// TIA Portal project "PLC_stage_DIPLOMA" (V19)

(* hardware
DEVICE "S7-1500/ET200MP station_1"  S7-1500 station
   slot 0: "Rail_0"  Rack  6ES7 590-1***0-0AA0
   slot 1: "PLC_1"  CPU 1513F-1 PN  6ES7 513-1FL02-0AB0  V2.9
      slot 3: "CPU display_1"  6ES7591-1AA00-0AA0
      slot 32768: "PROFINET interface_1"  X1
      slot 34817: "Virtual CP interface port_1"  Virtual CP interface port  Virtual CP interface port
   slot 2: "DI 32x24VDC HF_1"  DI 32x24VDC HF  6ES7 521-1BL00-0AB0  V2.2
   slot 3: "DQ 32x24VDC/0.5A HF_1"  DQ 32x24VDC/0.5A HF  6ES7 522-1BL01-0AB0  V1.1
   slot 4: "AI 8xU/I/RTD/TC ST_1"  AI 8xU/I/RTD/TC ST  6ES7 531-7KF00-0AB0  V2.2
DEVICE "ET 200SP station_1"  ET 200SP-Station
   slot 0: "Rack_0"  Rack  6ES5 710-8MAx1
   slot 0: "IO device_1"  IM 155-6 PN ST  6ES7 155-6AU01-0BN0  V4.2
   slot 1: "DI 8x24VDC ST_1"  DI 8x24VDC ST  6ES7 131-6BF01-0BA0  V0.0
      slot 1: "DI 8x24VDC ST_1"  DI 8x24VDC ST
   slot 2: "DI 8x24VDC ST_2"  DI 8x24VDC ST  6ES7 131-6BF01-0BA0  V0.0
      slot 1: "DI 8x24VDC ST_2"  DI 8x24VDC ST
   slot 3: "DQ 16x24VDC/0.5A ST_1"  DQ 16x24VDC/0.5A ST  6ES7 132-6BH01-0BA0  V0.0
      slot 1: "DQ 16x24VDC/0.5A ST_1"  DQ 16x24VDC/0.5A ST
   slot 4: "AI 4xU/I 2-wire ST_2"  AI 4xU/I 2-wire ST  6ES7 134-6HD01-0BA1  V2.0
      slot 1: "AI 4xU/I 2-wire ST_2"  AI 4xU/I 2-wire ST
   slot 5: "AQ 4xU/I ST_1"  AQ 4xU/I ST  6ES7 135-6HD00-0BA1  V1.1
      slot 1: "AQ 4xU/I ST_1"  AQ 4xU/I ST
   slot 6: "Server module_1"  Server module  6ES7 193-6PA00-0AA0  V1.1
      slot 1: "Server module_1"  Server module
   slot 127: "BA 2xRJ45"  BA 2xRJ45  6ES7 193-6AR00-0AA0  V0.0
      slot 1: "Port_1"  X1 P1 R  6ES7 193-6AR00-0AA0  V0.0
      slot 2: "Port_2"  X1 P2 R  6ES7 193-6AR00-0AA0  V0.0
DEVICE "PC-System_1"  SIMATIC PC station
   slot 0: "SIMATIC PC station"  Rail  SIMATIC PC-Station  V1.0
      slot 125: "Stationmanager"  Station_Manager  V6.0.4
   slot 1: "HMI_RT_2"  WinCC RT Advanced  6AV2 104-0xxxx-xxxx  17.0.0.0
      slot 33792: "Computer interface"  Host interface
   slot 2: "IE general_1"  IE General  IE_CP  V8.2.0
      slot 1: "PROFINET interface"  IEGeneral.Interface.8.2.0
DEVICE "HMI_1"  TP700 Comfort
   slot 0: "HMI_1"  TP700 Comfort  6AV2 124-0GC01-0AX0  17.0.0.0
   slot 1: "HMI_RT_1"  TP700 Comfort  6AV2 124-0GC01-0AX0  17.0.0.0
   slot 5: "HMI_1.IE_CP_1"  PROFINET Interface  17.0.0.0
      slot 1: "PROFINET Interface_1"  PROFINET Interface
         slot 1: "Port_1"  Port
         slot 2: "Port_2"  Port
   slot 7: "HMI_1.MPI/DP_CP_1"  MPI/DP Interface  17.0.0.0
*)

// ===== PLC "PLC_1"  CPU 1513F-1 PN =====

VAR_GLOBAL   // PLC tag table "additional_variables"
   "Get_value1_from_Matlab" AT %M11.0 : Bool;
   "AlwaysFALSE" AT %M0.3 : Bool;
   "Get_value2_from_Matlab" AT %M11.1 : Bool;
   "Send_value1_to_Matlab" AT %M11.2 : Bool;
   "Send_value2_to_Matlab" AT %M11.4 : Bool;
   "HMI_FN101_Visible1" AT %Q1.1 : Bool;
   "HMI_FN101_Visible2" AT %Q1.2 : Bool;
   "HMI_RB102_Visible" AT %Q1.4 : Bool;
   "HMI_WP101_Painted" AT %Q1.6 : Bool;
   "HMI_WP101_Visible" AT %M7.0 : Bool;
   "HMI_WP102_Visible" AT %M7.1 : Bool;
   "HMI_WP103_Visible" AT %M7.2 : Bool;
   "HMI_WP104_Visible" AT %M7.3 : Bool;
   "HMI_Main" AT %M7.4 : Bool;
   "HMI_PID" AT %M7.5 : Bool;
   "HMI_Status" AT %M7.6 : Bool;
   "Alarm_Collection" AT %MW21 : Int;
   "System_Byte" AT %MB0 : Byte;
   "tag3" AT %M4.0 : Bool;
   "check" AT %I2.4 : Bool;
   "HMI_PB_RB101" AT %M7.7 : Bool;
   "HMI_PB_RB102" AT %M8.0 : Bool;
   "HMI_PB_FN101" AT %M8.1 : Bool;
   "HMI_PB_CV101" AT %M8.2 : Bool;
END_VAR

VAR_GLOBAL   // PLC tag table "Main_variables"
   "RB-101" AT %Q0.0 : Bool;   // Spray Manipulator
   "CV-101" AT %Q4.0 : Bool;   // Conveyor
   "RB-102" AT %Q0.2 : Bool;   // Pick & Place Manipulator
   "FN-101" AT %M11.3 : Bool;   // Drying Fan
   "QI-101" AT %MW1 : Int;   // Package Counter
   "HMI_PS101" AT %M6.0 : Bool;   // Start process button in HMI
   "HMI_PS102" AT %M6.1 : Bool;   // Stop process button in HMI
   "HMI_ES101" AT %M6.2 : Bool;   // emergency button in HMI
   "HMI_PS103" AT %M6.3 : Bool;   // Automatic mode button in HMI
   "HMI_PS104" AT %M6.4 : Bool;   // Manual mode button in HMI
   "ALM_XA101_CV101" AT %M24.0 : Bool;   // ConveyorFault
   "ALM_XA103_RB101" AT %M24.1 : Bool;   // Spray ManipulatorFault
   "ALM_XA104_RB102" AT %M24.2 : Bool;   // Pick & Place ManipulatorFault
   "ALM_XA102_FN101" AT %M24.3 : Bool;   // FanFault
   "SIM_CV101" AT %M24.4 : Bool;   // ConveyorBroken
   "SIM_RB101" AT %M24.5 : Bool;   // Spray ManipulatorBroken
   "SIM_RB102" AT %M24.6 : Bool;   // Pick & Place ManipulatorBroken
   "SIM_FN101" AT %M24.7 : Bool;   // FanBroken
   "ZS-101" AT %I29.0 : Bool;   // Infeed Sensor
   "ZS-102" AT %I29.1 : Bool;   // Spray Position Sensor
   "ZS-103" AT %I29.2 : Bool;   // Drying/Fan Entry Sensor
   "ZS-104" AT %I29.3 : Bool;   // Pick&Place Position Sensor
   "PS101" AT %I0.0 : Bool;   // Start processbutton
   "PS102" AT %I0.1 : Bool;   // Stop process button
   "PS103" AT %I0.2 : Bool;   // Automatic mode button
   "PS104" AT %I0.3 : Bool;   // Manual mode button
   "ES101" AT %I0.4 : Bool;   // emergency button
END_VAR

VAR_GLOBAL CONSTANT   // PLC tag table "Main_variables"
   "None(1)" : Pip := 65535;
   "Automatic update(1)" : Pip := 0;
   "PIP 1(1)" : Pip := 1;
   "PIP 2(1)" : Pip := 2;
   "PIP 3(1)" : Pip := 3;
   "PIP 4(1)" : Pip := 4;
   "PIP 5(1)" : Pip := 5;
   "PIP 6(1)" : Pip := 6;
   "PIP 7(1)" : Pip := 7;
   "PIP 8(1)" : Pip := 8;
   "PIP 9(1)" : Pip := 9;
   "PIP 10(1)" : Pip := 10;
   "PIP 11(1)" : Pip := 11;
   "PIP 12(1)" : Pip := 12;
   "PIP 13(1)" : Pip := 13;
   "PIP 14(1)" : Pip := 14;
   "PIP 15(1)" : Pip := 15;
   "PIP 16(1)" : Pip := 16;
   "PIP 17(1)" : Pip := 17;
   "PIP 18(1)" : Pip := 18;
   "PIP 19(1)" : Pip := 19;
   "PIP 20(1)" : Pip := 20;
   "PIP 21(1)" : Pip := 21;
   "PIP 22(1)" : Pip := 22;
   "PIP 23(1)" : Pip := 23;
   "PIP 24(1)" : Pip := 24;
   "PIP 25(1)" : Pip := 25;
   "PIP 26(1)" : Pip := 26;
   "PIP 27(1)" : Pip := 27;
   "PIP 28(1)" : Pip := 28;
   "PIP 29(1)" : Pip := 29;
   "PIP 30(1)" : Pip := 30;
   "PIP 31(1)" : Pip := 31;
   "PIP OB Servo(1)" : Pip := 32768;
   "Local~MC(1)" : Hw_SubModule := 51;
   "Local~Common(1)" : Hw_SubModule := 50;
   "Local~Device(1)" : Hw_Device := 32;
   "Local~Configuration(1)" : Hw_SubModule := 33;
   "Local~Display(1)" : Hw_SubModule := 54;
   "Local~Exec(1)" : Hw_SubModule := 52;
   "Local(1)" : Hw_SubModule := 49;
   "Local~FExec(1)" : Hw_SubModule := 55;
   "Local~PROFINET_interface_1(1)" : Hw_Interface := 64;
   "Local~PROFINET_interface_1~Port_1(1)" : Hw_Interface := 65;
   "Local~PROFINET_interface_1~Port_2(1)" : Hw_Interface := 66;
   "Local~Virtual_communication_interface(1)" : Hw_Interface := 135;
   "Local~License_Manager(1)" : Hw_SubModule := 42;
   "OB_Main(1)" : OB_PCYCLE := 1;
   "OB_FOB_RTG1" : OB_Cyclic := 123;
   "Local~DI_32x24VDC_HF_1(1)" : Hw_SubModule := 257;
   "Local~DQ_32x24VDC_0_5A_HF_1(1)" : Hw_SubModule := 258;
   "Local~AI_8xU_I_HS_1" : Hw_SubModule := 259;
   "Local~AQ_8xU_I_HS_1" : Hw_SubModule := 260;
END_VAR

DATA_BLOCK "Block_1_DB"   // DB12
{ S7_Optimized_Access := 'TRUE' }
VERSION : 0.1
// stored: InstanceOfName Auto_mode
"Auto_mode"
BEGIN
END_DATA_BLOCK

DATA_BLOCK "Manu_mode_DB"   // DB13
{ S7_Optimized_Access := 'TRUE' }
VERSION : 0.1
// stored: InstanceOfName Manu_mode
"Manu_mode"
BEGIN
END_DATA_BLOCK

// folder: System blocks/Program resources

DATA_BLOCK "IEC_Timer_0_DB_3"   // DB3
{ S7_Optimized_Access := 'TRUE' }
AUTHOR : Simatic
FAMILY : IEC
NAME : IEC_TMR
VERSION : 1.0
// stored: InstanceOfName IEC_TIMER
"IEC_TIMER"
BEGIN
END_DATA_BLOCK

DATA_BLOCK "IEC_Timer_0_DB"   // DB4
{ S7_Optimized_Access := 'TRUE' }
AUTHOR : Simatic
FAMILY : IEC
NAME : IEC_TMR
VERSION : 1.0
// stored: InstanceOfName IEC_TIMER
"IEC_TIMER"
BEGIN
END_DATA_BLOCK

DATA_BLOCK "IEC_Timer_0_DB_1"   // DB6
{ S7_Optimized_Access := 'TRUE' }
AUTHOR : Simatic
FAMILY : IEC
NAME : IEC_TMR
VERSION : 1.0
// stored: InstanceOfName IEC_TIMER
"IEC_TIMER"
BEGIN
END_DATA_BLOCK

DATA_BLOCK "IEC_Timer_0_DB_2"   // DB7
{ S7_Optimized_Access := 'TRUE' }
AUTHOR : Simatic
FAMILY : IEC
NAME : IEC_TMR
VERSION : 1.0
// stored: InstanceOfName IEC_TIMER
"IEC_TIMER"
BEGIN
END_DATA_BLOCK

DATA_BLOCK "IEC_Timer_0_DB_4"   // DB10
{ S7_Optimized_Access := 'TRUE' }
AUTHOR : Simatic
FAMILY : IEC
NAME : IEC_TMR
VERSION : 1.0
// stored: InstanceOfName IEC_TIMER
"IEC_TIMER"
BEGIN
END_DATA_BLOCK

DATA_BLOCK "IEC_Counter_0_DB_2"   // DB11
{ S7_Optimized_Access := 'TRUE' }
AUTHOR : Simatic
FAMILY : IEC
NAME : CNTR
VERSION : 1.0
// stored: InstanceOfName IEC_COUNTER
"IEC_COUNTER"
BEGIN
END_DATA_BLOCK

// folder: (top level)

FUNCTION_BLOCK "Auto_mode"   // FB2, LAD
{ S7_Optimized_Access := 'TRUE' }
VERSION : 0.1
   VAR_TEMP   // added for the SCL form of the ladder/FBD networks
      _w1 : Bool;
      _w2 : Bool;
      _w3 : Bool;
      _w4 : Bool;
   END_VAR
BEGIN

REGION Network 1: Auto
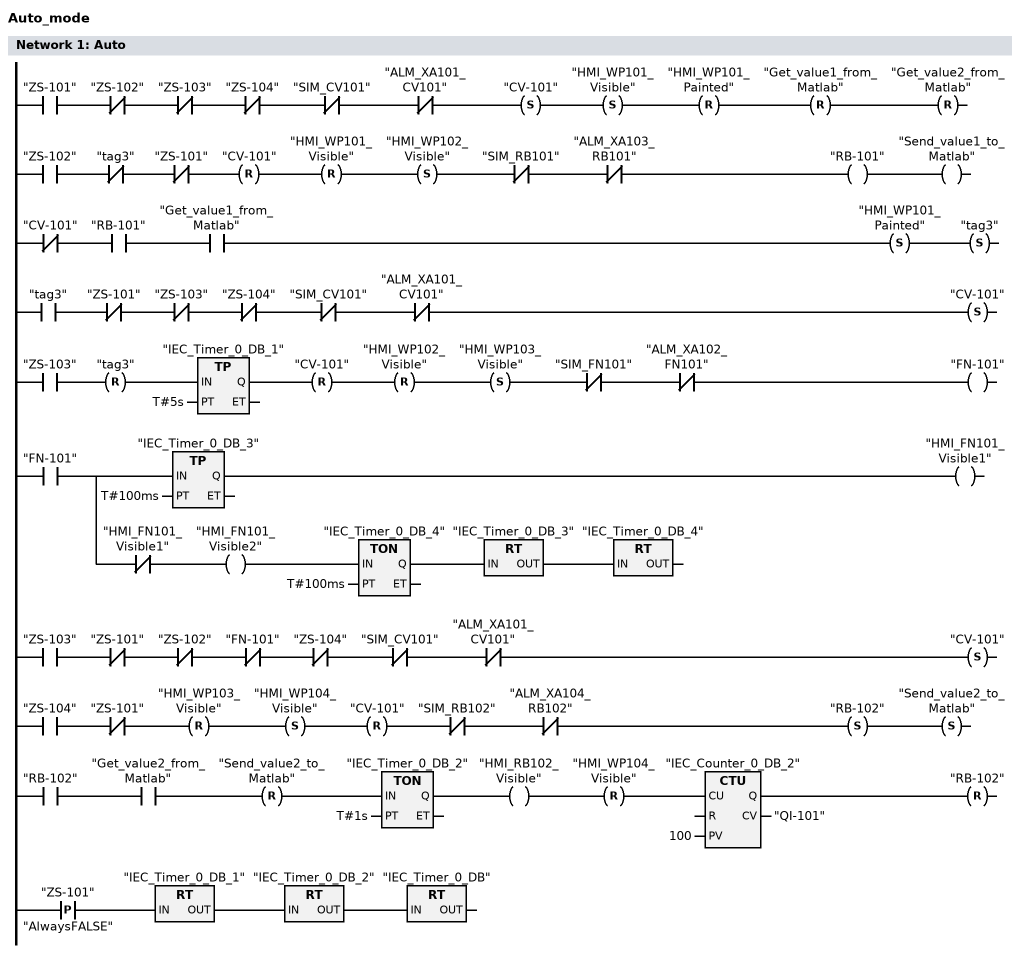
   IF "ZS-101" AND NOT "ZS-102" AND NOT "ZS-103" AND NOT "ZS-104" AND NOT "SIM_CV101" AND NOT "ALM_XA101_CV101" THEN
       "CV-101" := TRUE;
       "HMI_WP101_Visible" := TRUE;
       "HMI_WP101_Painted" := FALSE;
       "Get_value1_from_Matlab" := FALSE;
       "Get_value2_from_Matlab" := FALSE;
   END_IF;
   #_w1 := "ZS-102" AND NOT "tag3" AND NOT "ZS-101";
   IF #_w1 THEN
       "CV-101" := FALSE;
       "HMI_WP101_Visible" := FALSE;
       "HMI_WP102_Visible" := TRUE;
   END_IF;
   "RB-101" := #_w1 AND NOT "SIM_RB101" AND NOT "ALM_XA103_RB101";
   "Send_value1_to_Matlab" := "RB-101";
   IF NOT "CV-101" AND "RB-101" AND "Get_value1_from_Matlab" THEN
       "HMI_WP101_Painted" := TRUE;
       "tag3" := TRUE;
   END_IF;
   IF "tag3" AND NOT "ZS-101" AND NOT "ZS-103" AND NOT "ZS-104" AND NOT "SIM_CV101" AND NOT "ALM_XA101_CV101" THEN
       "CV-101" := TRUE;
   END_IF;
   IF "ZS-103" THEN "tag3" := FALSE; END_IF;
   "IEC_Timer_0_DB_1".TP(IN := "ZS-103", PT := T#5s);
   IF "IEC_Timer_0_DB_1".Q THEN
       "CV-101" := FALSE;
       "HMI_WP102_Visible" := FALSE;
       "HMI_WP103_Visible" := TRUE;
   END_IF;
   "FN-101" := "IEC_Timer_0_DB_1".Q AND NOT "SIM_FN101" AND NOT "ALM_XA102_FN101";
   "IEC_Timer_0_DB_3".TP(IN := "FN-101", PT := T#100ms);
   "HMI_FN101_Visible1" := "IEC_Timer_0_DB_3".Q;
   "HMI_FN101_Visible2" := "FN-101" AND NOT "HMI_FN101_Visible1";
   "IEC_Timer_0_DB_4".TON(IN := "HMI_FN101_Visible2", PT := T#100ms);
   IF "IEC_Timer_0_DB_4".Q THEN
       RESET_TIMER("IEC_Timer_0_DB_3");
       RESET_TIMER("IEC_Timer_0_DB_4");
   END_IF;
   IF "ZS-103" AND NOT "ZS-101" AND NOT "ZS-102" AND NOT "FN-101" AND NOT "ZS-104" AND NOT "SIM_CV101" AND NOT "ALM_XA101_CV101" THEN
       "CV-101" := TRUE;
   END_IF;
   #_w2 := "ZS-104" AND NOT "ZS-101";
   IF #_w2 THEN
       "HMI_WP103_Visible" := FALSE;
       "HMI_WP104_Visible" := TRUE;
       "CV-101" := FALSE;
   END_IF;
   IF #_w2 AND NOT "SIM_RB102" AND NOT "ALM_XA104_RB102" THEN
       "RB-102" := TRUE;
       "Send_value2_to_Matlab" := TRUE;
   END_IF;
   #_w3 := "RB-102" AND "Get_value2_from_Matlab";
   IF #_w3 THEN "Send_value2_to_Matlab" := FALSE; END_IF;
   "IEC_Timer_0_DB_2".TON(IN := #_w3, PT := T#1s);
   "HMI_RB102_Visible" := "IEC_Timer_0_DB_2".Q;
   IF "IEC_Timer_0_DB_2".Q THEN "HMI_WP104_Visible" := FALSE; END_IF;
   "IEC_Counter_0_DB_2".CTU(CU := "IEC_Timer_0_DB_2".Q, PV := 100, CV => "QI-101");
   IF "IEC_Counter_0_DB_2".Q THEN "RB-102" := FALSE; END_IF;
   #_w4 := "ZS-101" AND NOT "AlwaysFALSE";   // rising edge of "ZS-101"
   "AlwaysFALSE" := "ZS-101";
   IF #_w4 THEN
       RESET_TIMER("IEC_Timer_0_DB_1");
       RESET_TIMER("IEC_Timer_0_DB_2");
       RESET_TIMER("IEC_Timer_0_DB");
   END_IF;
END_REGION
END_FUNCTION_BLOCK

FUNCTION_BLOCK "Manu_mode"   // FB3, LAD
{ S7_Optimized_Access := 'TRUE' }
VERSION : 0.1
   VAR_TEMP   // added for the SCL form of the ladder/FBD networks
      _w1 : Bool;
      _w2 : Bool;
   END_VAR
BEGIN

REGION Network 1: Manu
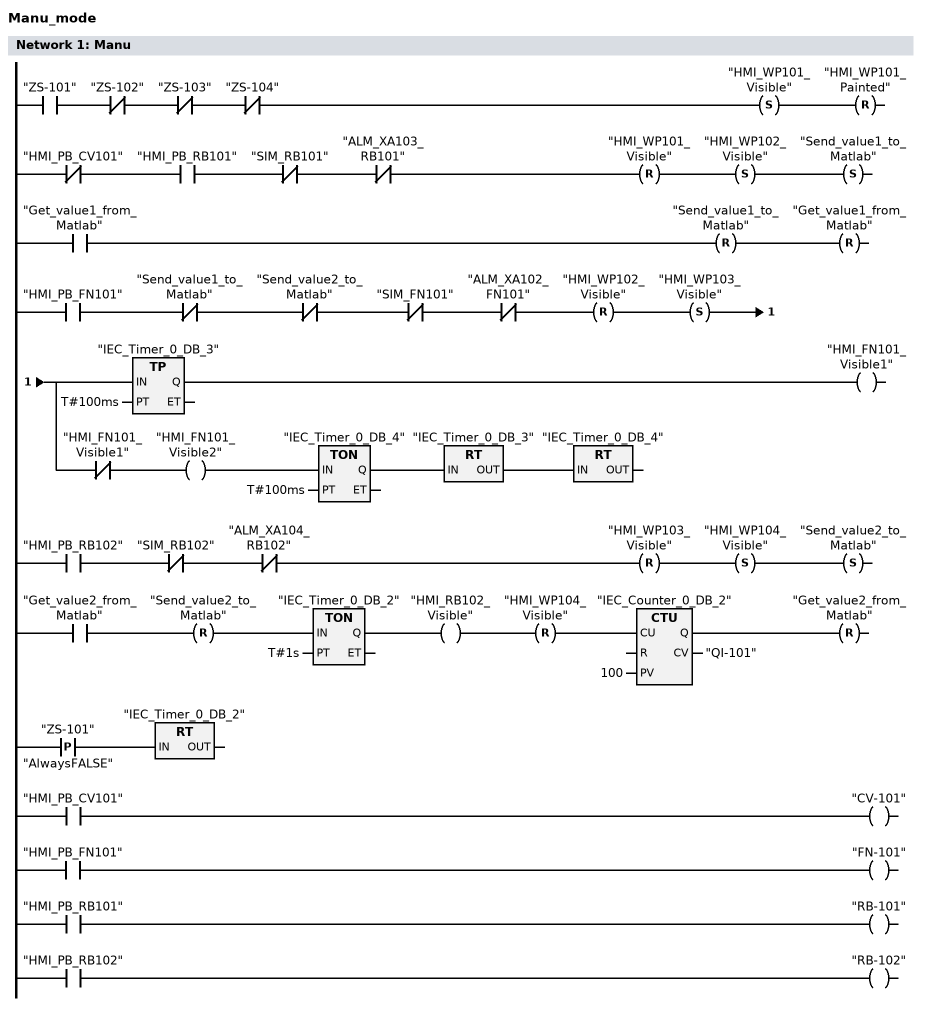
   IF "ZS-101" AND NOT "ZS-102" AND NOT "ZS-103" AND NOT "ZS-104" THEN
       "HMI_WP101_Visible" := TRUE;
       "HMI_WP101_Painted" := FALSE;
   END_IF;
   IF NOT "HMI_PB_CV101" AND "HMI_PB_RB101" AND NOT "SIM_RB101" AND NOT "ALM_XA103_RB101" THEN
       "HMI_WP101_Visible" := FALSE;
       "HMI_WP102_Visible" := TRUE;
       "Send_value1_to_Matlab" := TRUE;
   END_IF;
   IF "Get_value1_from_Matlab" THEN
       "Send_value1_to_Matlab" := FALSE;
       "Get_value1_from_Matlab" := FALSE;
   END_IF;
   #_w1 := "HMI_PB_FN101" AND NOT "Send_value1_to_Matlab" AND NOT "Send_value2_to_Matlab" AND NOT "SIM_FN101" AND NOT "ALM_XA102_FN101";
   IF #_w1 THEN
       "HMI_WP102_Visible" := FALSE;
       "HMI_WP103_Visible" := TRUE;
   END_IF;
   "IEC_Timer_0_DB_3".TP(IN := #_w1, PT := T#100ms);
   "HMI_FN101_Visible1" := "IEC_Timer_0_DB_3".Q;
   "HMI_FN101_Visible2" := #_w1 AND NOT "HMI_FN101_Visible1";
   "IEC_Timer_0_DB_4".TON(IN := "HMI_FN101_Visible2", PT := T#100ms);
   IF "IEC_Timer_0_DB_4".Q THEN
       RESET_TIMER("IEC_Timer_0_DB_3");
       RESET_TIMER("IEC_Timer_0_DB_4");
   END_IF;
   IF "HMI_PB_RB102" AND NOT "SIM_RB102" AND NOT "ALM_XA104_RB102" THEN
       "HMI_WP103_Visible" := FALSE;
       "HMI_WP104_Visible" := TRUE;
       "Send_value2_to_Matlab" := TRUE;
   END_IF;
   IF "Get_value2_from_Matlab" THEN "Send_value2_to_Matlab" := FALSE; END_IF;
   "IEC_Timer_0_DB_2".TON(IN := "Get_value2_from_Matlab", PT := T#1s);
   "HMI_RB102_Visible" := "IEC_Timer_0_DB_2".Q;
   IF "IEC_Timer_0_DB_2".Q THEN "HMI_WP104_Visible" := FALSE; END_IF;
   "IEC_Counter_0_DB_2".CTU(CU := "IEC_Timer_0_DB_2".Q, PV := 100, CV => "QI-101");
   IF "IEC_Counter_0_DB_2".Q THEN "Get_value2_from_Matlab" := FALSE; END_IF;
   #_w2 := "ZS-101" AND NOT "AlwaysFALSE";   // rising edge of "ZS-101"
   "AlwaysFALSE" := "ZS-101";
   IF #_w2 THEN RESET_TIMER("IEC_Timer_0_DB_2"); END_IF;
   "CV-101" := "HMI_PB_CV101";
   "FN-101" := "HMI_PB_FN101";
   "RB-101" := "HMI_PB_RB101";
   "RB-102" := "HMI_PB_RB102";
END_REGION
END_FUNCTION_BLOCK

ORGANIZATION_BLOCK "Main"   // OB1, LAD, ProgramCycle
TITLE = "Main Program Sweep (Cycle)"
{ S7_Optimized_Access := 'TRUE' }
VERSION : 0.1
   VAR_INPUT
      Initial_Call : Bool;   // Initial call of this OB
      Remanence : Bool;   // =True, if remanent data are available
   END_VAR
BEGIN

REGION Network 1
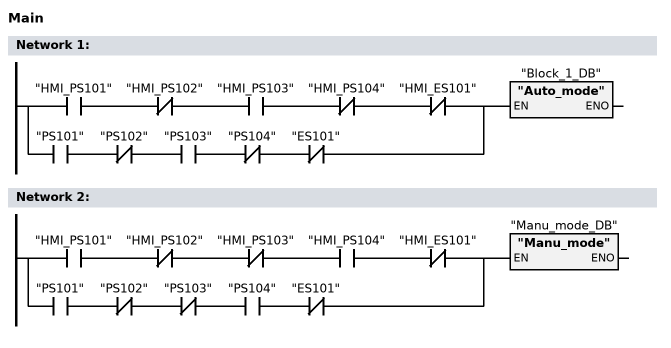
   RUNG wire#powerrail
      Contact( "HMI_PS101" )
      I_Contact( "HMI_PS102" )
      Contact( "HMI_PS103" )
      I_Contact( "HMI_PS104" )
      I_Contact( "HMI_ES101" )
      wire#w1
      "Block_1_DB"()
   END_RUNG
   RUNG wire#powerrail
      Contact( "PS101" )
      I_Contact( "PS102" )
      Contact( "PS103" )
      I_Contact( "PS104" )
      I_Contact( "ES101" )
   END_RUNG wire#w1
   // the same network as SCL:
   IF ("HMI_PS101" AND NOT "HMI_PS102" AND "HMI_PS103" AND NOT "HMI_PS104" AND NOT "HMI_ES101") OR ("PS101" AND NOT "PS102" AND "PS103" AND NOT "PS104" AND NOT "ES101") THEN
       "Block_1_DB"();   // "Auto_mode"
   END_IF;
END_REGION

REGION Network 2
   RUNG wire#powerrail
      Contact( "HMI_PS101" )
      I_Contact( "HMI_PS102" )
      I_Contact( "HMI_PS103" )
      Contact( "HMI_PS104" )
      I_Contact( "HMI_ES101" )
      wire#w1
      "Manu_mode_DB"()
   END_RUNG
   RUNG wire#powerrail
      Contact( "PS101" )
      I_Contact( "PS102" )
      I_Contact( "PS103" )
      Contact( "PS104" )
      I_Contact( "ES101" )
   END_RUNG wire#w1
   // the same network as SCL:
   IF ("HMI_PS101" AND NOT "HMI_PS102" AND NOT "HMI_PS103" AND "HMI_PS104" AND NOT "HMI_ES101") OR ("PS101" AND NOT "PS102" AND NOT "PS103" AND "PS104" AND NOT "ES101") THEN
       "Manu_mode_DB"();   // "Manu_mode"
   END_IF;
END_REGION
END_ORGANIZATION_BLOCK

(* ===== HMI "HMI_RT_2" =====
system functions are stored by id; their names below are inferred from use
connection "HMI_Connection_2": ETHERNET, S7_1500_OMS
connection "HMI_Connection_3": ETHERNET, S7_1500_OMS

HMI tags "Default tag table"
   "HMI_FN101_Visible1" : Bool = PLC HMI_FN101_Visible1 AT %Q1.1, 1 s
   "HMI_FN101_Visible2" : Bool = PLC HMI_FN101_Visible2 AT %Q1.2, 1 s
   "ZS-101" : Bool = PLC "ZS-101" AT %I29.0, 1 s
   "ZS-102" : Bool = PLC "ZS-102" AT %I29.1, 1 s
   "ZS-103" : Bool = PLC "ZS-103" AT %I29.2, 1 s
   "ZS-104" : Bool = PLC "ZS-104" AT %I29.3, 1 s
   "RB-101" : Bool = PLC "RB-101" AT %Q0.0, 1 s
   "FAN" : Bool = PLC "FN-101" AT %M11.3, 1 s
   "CV-101" : Bool = PLC "CV-101" AT %Q4.0, 1 s
   "RB-102" : Bool = PLC "RB-102" AT %Q0.2, 1 s
   "HMI_RB102_Visible" : Bool = PLC HMI_RB102_Visible AT %Q1.4, 1 s
   "amount" : Int = PLC "QI-101" AT %MW1, 1 s
   "block_color" : Bool = PLC HMI_WP101_Painted AT %Q1.6, 1 s
   "start" : Bool = PLC HMI_PS101 AT %M6.0, 1 s
   "HMI_WP101_Visible" : Bool = PLC HMI_WP101_Visible AT %M7.0, 1 s
   "emergency" : Bool = PLC HMI_ES101 AT %M6.2, 1 s
   "stop" : Bool = PLC HMI_PS102 AT %M6.1, 1 s
   "auto" : Bool = PLC HMI_PS103 AT %M6.3, 1 s
   "manu" : Bool = PLC HMI_PS104 AT %M6.4, 1 s
   "Alarm_Collection" : Int = PLC Alarm_Collection AT %MW21, 1 s
   "manip1_error" : Bool = PLC ALM_XA103_RB101 AT %M24.1, 1 s
   "manip1_broken" : Bool = PLC SIM_RB101 AT %M24.5, 1 s
   "fan_error" : Bool = PLC ALM_XA102_FN101 AT %M24.3, 1 s
   "fan_broken" : Bool = PLC SIM_FN101 AT %M24.7, 1 s
   "conv_broken" : Bool = PLC SIM_CV101 AT %M24.4, 1 s
   "conv_error" : Bool = PLC ALM_XA101_CV101 AT %M24.0, 1 s
   "manip2_error" : Bool = PLC ALM_XA104_RB102 AT %M24.2, 1 s
   "manip2_broken" : Bool = PLC SIM_RB102 AT %M24.6, 1 s
   "check" : Bool = PLC check AT %I2.4, 1 s
   "HMI_WP102_Visible" : Bool = PLC HMI_WP102_Visible AT %M7.1, 1 s
   "HMI_WP103_Visible" : Bool = PLC HMI_WP103_Visible AT %M7.2, 1 s
   "HMI_WP104_Visible" : Bool = PLC HMI_WP104_Visible AT %M7.3, 1 s
   "HMI_Main" : Bool = PLC HMI_Main AT %M7.4, 1 s
   "HMI_PID" : Bool = PLC HMI_PID AT %M7.5, 1 s
   "HMI_Status" : Bool = PLC HMI_Status AT %M7.6, 1 s
   "HMI_PB_RB101" : Bool = PLC HMI_PB_RB101 AT %M7.7, 1 s
   "HMI_PB_FN101" : Bool = PLC HMI_PB_FN101 AT %M8.1, 1 s
   "HMI_PB_RB102" : Bool = PLC HMI_PB_RB102 AT %M8.0, 1 s
   "HMI_PB_CV101" : Bool = PLC HMI_PB_CV101 AT %M8.2, 1 s

discrete alarms
   1: 'Something is wrong with the conveyor!!!', class Errors, trigger "Alarm_Collection" bit 0
   2: 'Conveyor is in tech-service.', class Warnings, trigger "Alarm_Collection" bit 1
   3: 'Something is wrong with the Manipulator 1!!!', class Errors, trigger "Alarm_Collection" bit 2
   4: 'Manipulator 1 is in tech-service.', class Warnings, trigger "Alarm_Collection" bit 3
   5: 'Something is wrong with the Fan!!!', class Errors, trigger "Alarm_Collection" bit 4
   6: 'Fan is in tech-service.', class Warnings, trigger "Alarm_Collection" bit 5
   7: 'Something is wrong with the Manipulator 2!!!', class Errors, trigger "Alarm_Collection" bit 6
   8: 'Manipulator 2 is in tech-service.', class Warnings, trigger "Alarm_Collection" bit 7

text list "OFF_ON_LIST": 0 ''; 1 ''

screen "Main Part" 1980x1080
   Circle "Circle_6" at 216,721 size 41x41
      Appearance <- "RB-101"
   IOField "I/O field_1" at 1077,716 size 145x38; FormatPattern s99999
      ProcessValue <- "amount"
   Circle "Circle_7" at 1051,213 size 41x41
      Appearance <- "RB-102"
   TextField "Text field_1" at 268,778 size 107x37; Text 'RB-101'
   TextField "Text field_2" at 569,707 size 105x37; Text 'FN-101'
   TextField "Text field_3" at 1098,771 size 102x37; Text 'QI-101'
   TextField "Text field_4" at 1094,165 size 107x37; Text 'RB-102'
   TextField "Text field_6" at 111,158 size 108x39; Text 'ZS-101'
   TextField "Text field_5" at 262,158 size 108x39; Text 'ZS-102'
   TextField "Text field_7" at 396,158 size 108x39; Text 'ZS-103'
   TextField "Text field_8" at 818,159 size 108x39; Text 'ZS-104'
   Button "Button_2" at 1360,176 size 190x61; TextOff 'Start'; TextList "OFF_ON_LIST"
      on Press: SetBit("start"); ResetBit("stop")
      ProcessValue <- "start"
   Button "Button_6" at 1360,264 size 190x61; TextOff 'STOP'
      on Press: SetBit("stop"); ResetBit("start")
      on Release: ResetBit("stop")
   GraphicView "Graphic view_2" at 375,721 size 49x47; Picture "Graphic_7"
      Visibility <- "manip1_broken"
   GraphicView "Graphic view_3" at 293,721 size 49x47; Picture "Graphic_8"
      Visibility <- "manip1_error"
   GraphicView "Graphic view_5" at 1199,213 size 49x47; Picture "Graphic_7"
      Appearance <- "manip2_broken"
   GraphicView "Graphic view_7" at 1124,212 size 49x47; Picture "Graphic_8"
      Appearance <- "manip2_error"
   Circle "Circle_16" at 147,213 size 29x29
      Appearance <- "ZS-101"
   Circle "Circle_18" at 298,211 size 29x29
      Appearance <- "ZS-102"
   Circle "Circle_20" at 758,488 size 41x41
      Appearance <- "CV-101"
   GraphicView "Graphic view_1" at 832,488 size 49x47; Picture "Graphic_8"
      Appearance <- "conv_error"
   GraphicView "Graphic view_8" at 904,488 size 49x47; Picture "Graphic_7"
      Appearance <- "conv_broken"
   TextField "Text field_11" at 815,544 size 104x37; Text 'CV-101'
   Circle "Circle_8" at 455,210 size 29x29
      Appearance <- "ZS-103"
   Circle "Circle_9" at 858,208 size 29x29
      Appearance <- "ZS-104"
   Rectangle "Rectangle_15" at 1100,329 size 76x141
      Visibility <- "HMI_RB102_Visible"
   Rectangle "Rectangle_18" at 1116,472 size 49x109
      Visibility <- "HMI_RB102_Visible"
   Rectangle "Rectangle_19" at 1109,580 size 64x24
      Visibility <- "HMI_RB102_Visible"
   Group "Group" at 128,304 size 110x99
   Circle "Circle_11" at 523,652 size 41x41
      Appearance <- "FAN"
   GraphicView "Graphic view_4" at 658,651 size 49x47; Picture "Graphic_7"
      Appearance <- "fan_broken"
   GraphicView "Graphic view_6" at 592,651 size 49x47; Picture "Graphic_8"
      Appearance <- "fan_error"
   Circle "Circle_13" at 1723,542 size 90x90
      Appearance <- "emergency"
   Button "Button_12" at 1363,555 size 190x61; TextOff 'Emergency'
      on Press: SetBit("emergency"); ResetBit("start"); ResetBit("auto"); ResetBit("manu")
      on Release: ResetBit("emergency")
   Button "Button_1" at 1357,440 size 190x61; TextOff 'Auto Mode'
      on Press: SetBit("auto"); ResetBit("manu")
   Button "Button_13" at 1358,354 size 190x61; TextOff 'Manu Mode'
      on Press: SetBit("manu"); ResetBit("auto")
   Button "Button_14" at 1653,175 size 190x61; TextOff 'PB_RB101'
      on Press: SetBit("HMI_PB_RB101")
      on Release: ResetBit("HMI_PB_RB101")
   Button "Button_3" at 1653,348 size 190x61; TextOff 'PB_RB102'
      on Press: SetBit("HMI_PB_RB102")
      on Release: ResetBit("HMI_PB_RB102")
   Button "Button_4" at 1653,259 size 190x61; TextOff 'PB_FN101'
      on Press: SetBit("HMI_PB_FN101")
      on Release: ResetBit("HMI_PB_FN101")
   Button "Button_5" at 1654,430 size 190x61; TextOff 'PB_CV101'
      on Press: SetBit("HMI_PB_CV101")
      on Release: ResetBit("HMI_PB_CV101")
   GraphicView "Graphic view_15" at 293,721 size 49x47; Picture "Graphic_10"
      Visibility <- "manip1_error"
   GraphicView "Graphic view_16" at 375,721 size 49x47; Picture "Graphic_9"
      Visibility <- "manip1_broken"
   GraphicView "Graphic view_17" at 592,651 size 49x47; Picture "Graphic_10"
      Visibility <- "fan_error"
   GraphicView "Graphic view_18" at 658,651 size 49x47; Picture "Graphic_9"
      Visibility <- "fan_broken"
   GraphicView "Graphic view_19" at 904,488 size 49x47; Picture "Graphic_9"
      Visibility <- "conv_broken"
   GraphicView "Graphic view_20" at 832,488 size 49x47; Picture "Graphic_10"
      Visibility <- "conv_error"
   GraphicView "Graphic view_21" at 1124,212 size 49x47; Picture "Graphic_10"
      Visibility <- "manip2_error"
   GraphicView "Graphic view_22" at 1199,213 size 49x47; Picture "Graphic_9"
      Visibility <- "manip2_broken"
   TextField "Text field_10" at 1507,25 size 21x33; Text 'Text'
   Button "Button_7" at 1338,26 size 536x43; TextOff 'CONTROL PANEL'
      on Press: SetBit("HMI_Main")
      Appearance <- "HMI_Main"
   Button "Button_8" at 1338,68 size 536x43; TextOff 'PID'
      on Press: ResetBit("HMI_Main"); ActivateScreen("PID", 0)
      Visibility <- "HMI_Main"
   Button "Button_9" at 1338,110 size 536x43; TextOff 'ERROR STATUS'
      on Press: ResetBit("HMI_Main"); ActivateScreen("Error_Status", 0)
      Visibility <- "HMI_Main"
   Group "Group_1" at 269,304 size 110x99
   Group "Group_2" at 472,303 size 110x99
   Group "Group_3" at 843,305 size 110x99
   Rectangle "Rectangle_22" at 1031,329 size 147x73
      Visibility <- "HMI_RB102_Visible"
   Rectangle "Rectangle_23" at 918,340 size 113x47
      Visibility <- "HMI_RB102_Visible"
   Rectangle "Rectangle_24" at 893,333 size 25x61
      Visibility <- "HMI_RB102_Visible"
   GraphicView "Graphic view_9" at 551,197 size 129x125; Picture "Graphic_14"
      Visibility <- "FAN"
   GraphicView "Graphic view_10" at 551,198 size 129x125; Picture "Graphic_15"
      Visibility <- "HMI_FN101_Visible1"
   GraphicView "Graphic view_11" at 551,353 size 129x125; Picture "Graphic_14"
   GraphicView "Graphic view_12" at 551,353 size 129x125; Picture "Graphic_15"
      Visibility <- "HMI_FN101_Visible1"
   GraphicView "Graphic view_13" at 551,198 size 129x125; Picture "Graphic_16"
      Visibility <- "HMI_FN101_Visible2"
   GraphicView "Graphic view_14" at 551,353 size 129x125; Picture "Graphic_16"
      Visibility <- "HMI_FN101_Visible2"
   TextField "Text field_12" at 1717,635 size 102x37; Text 'ES-101'
   Rectangle "Rectangle_44" at 128,304 size 110x74
      Appearance <- "block_color"
      Visibility <- "HMI_WP101_Visible"
   Rectangle "Rectangle_45" at 128,378 size 110x25
      Appearance <- "block_color"
      Visibility <- "HMI_WP101_Visible"
   Rectangle "Rectangle_31" at 269,304 size 110x74
      Appearance <- "block_color"
      Visibility <- "HMI_WP102_Visible"
   Rectangle "Rectangle_32" at 269,378 size 110x25
      Appearance <- "block_color"
      Visibility <- "HMI_WP102_Visible"
   Rectangle "Rectangle_33" at 472,303 size 110x74
      Appearance <- "block_color"
      Visibility <- "HMI_WP103_Visible"
   Rectangle "Rectangle_34" at 472,377 size 110x25
      Appearance <- "block_color"
      Visibility <- "HMI_WP103_Visible"
   Rectangle "Rectangle_35" at 843,305 size 110x74
      Appearance <- "block_color"
      Visibility <- "HMI_WP104_Visible"
   Rectangle "Rectangle_46" at 843,379 size 110x25
      Appearance <- "block_color"
      Visibility <- "HMI_WP104_Visible"

screen "Error_Status" 1980x1080
   AlarmView "Alarm view_1" at 231,25 size 1070x685
   Button "Button_17" at 1431,170 size 347x43; TextOff 'ALM_XA101_ConveyorFault'
      on Press: function_b3f726e6("Alarm_Collection", 0); SetBit("conv_error")
   Button "Button_18" at 1485,410 size 248x43; TextOff 'SIM_CV101_Broken'
      on Press: function_b3f726e6("Alarm_Collection", 1); SetBit("conv_broken")
   Button "Button_20" at 1431,290 size 347x43; TextOff 'ALM_XA103_RB101Fault'
      on Press: function_b3f726e6("Alarm_Collection", 2); SetBit("manip1_error")
   Button "Button_22" at 1485,530 size 248x43; TextOff 'SIM_RB101_Broken'
      on Press: function_b3f726e6("Alarm_Collection", 3); SetBit("manip1_broken")
   Button "Button_19" at 1432,230 size 347x43; TextOff 'ALM_XA102_FanFault'
      on Press: function_b3f726e6("Alarm_Collection", 4); SetBit("fan_error")
   Button "Button_23" at 1485,470 size 248x43; TextOff 'SIM_FN101_Broken'
      on Press: function_b3f726e6("Alarm_Collection", 5); SetBit("fan_broken")
   Button "Button_24" at 1430,350 size 347x43; TextOff 'ALM_XA104_RB102Fault'
      on Press: function_b3f726e6("Alarm_Collection", 6); SetBit("manip2_error")
   Button "Button_25" at 1485,590 size 248x43; TextOff 'SIM_RB102_Broken'
      on Press: function_b3f726e6("Alarm_Collection", 7); SetBit("manip2_broken")
   Button "Button_7" at 1485,650 size 248x43; TextOff 'Repair all'
      on Press: function_a9b64e44("Alarm_Collection", 0); function_a9b64e44("Alarm_Collection", 1); function_a9b64e44("Alarm_Collection", 2); function_a9b64e44("Alarm_Collection", 3); function_a9b64e44("Alarm_Collection", 4); function_a9b64e44("Alarm_Collection", 5); function_a9b64e44("Alarm_Collection", 6); function_a9b64e44("Alarm_Collection", 7); ResetBit("conv_error"); ResetBit("conv_broken"); ResetBit("manip1_error"); ResetBit("manip1_broken"); ResetBit("fan_error"); ResetBit("fan_broken"); ResetBit("manip2_error"); ResetBit("manip2_broken")
   TextField "Text field_10" at 1507,25 size 21x33; Text 'Text'
   Button "Button_1" at 1338,26 size 536x43; TextOff 'ERROR STATUS'
      on Press: SetBit("HMI_Status")
      Appearance <- "HMI_Status"
   Button "Button_8" at 1338,68 size 536x43; TextOff 'PID'
      on Press: ResetBit("HMI_Status"); ActivateScreen("PID", 0)
      Visibility <- "HMI_Status"
   Button "Button_9" at 1338,110 size 536x43; TextOff 'CONTROL PANEL'
      on Press: ResetBit("HMI_Status"); ActivateScreen("Main Part", 0)
      Visibility <- "HMI_Status"

screen "PID" 1980x1080
   TextField "Text field_10" at 1507,25 size 21x33; Text 'Text'
   Button "Button_1" at 1338,26 size 536x43; TextOff 'PID'
      on Press: SetBit("HMI_PID")
      Appearance <- "HMI_PID"
   Button "Button_8" at 1338,68 size 536x43; TextOff 'ERROR STATUS'
      on Press: ResetBit("HMI_PID"); ActivateScreen("Error_Status", 0)
      Visibility <- "HMI_PID"
   Button "Button_9" at 1338,110 size 536x43; TextOff 'CONTROL PANEL'
      on Press: ResetBit("HMI_PID"); ActivateScreen("Main Part", 0)
      Visibility <- "HMI_PID"
   TrendView "Trend view_1" at 231,25 size 1070x685
   IOField "I/O field_1" at 1704,194 size 145x38; FormatPattern s99999
      ProcessValue <- "amount"
   IOField "I/O field_2" at 1704,262 size 145x38; FormatPattern s99999
      ProcessValue <- "amount"
   IOField "I/O field_3" at 1704,330 size 145x38; FormatPattern s99999
      ProcessValue <- "amount"
   IOField "I/O field_4" at 1704,398 size 145x38; FormatPattern s99999
      ProcessValue <- "amount"
   TextField "Text field_4" at 1570,194 size 119x37; Text 'Setpoint'
   TextField "Text field_1" at 1628,262 size 58x37; Text 'K_p'
   TextField "Text field_2" at 1628,330 size 49x37; Text 'K_i'
   TextField "Text field_3" at 1628,398 size 58x37; Text 'K_d'
   Rectangle "Rectangle_22" at 1364,206 size 174x218
      Visibility <- "HMI_RB102_Visible"
   Circle "Circle_13" at 1461,226 size 63x63
      Appearance <- "emergency"
   Circle "Circle_1" at 1461,337 size 63x63
      Appearance <- "emergency"
   TextField "Text field_5" at 1374,237 size 72x37; Text 'Start'
   TextField "Text field_6" at 1375,348 size 67x37; Text 'Stop'
*)

(* ===== HMI "HMI_RT_1" =====
system functions are stored by id; their names below are inferred from use
connection "HMI_Connection_4": ETHERNET, S7_1500_OMS

HMI tags "Default tag table"
   "Tag_ScreenNumber" : UInt, internal
   "Alarm_Collection" : Int = PLC Alarm_Collection AT %MW21, 1 s
   "amount" : Int = PLC "QI-101" AT %MW1, 1 s
   "auto" : Bool = PLC HMI_PS103 AT %M6.3, 1 s
   "block_color" : Bool = PLC HMI_WP101_Painted AT %Q1.6, 1 s
   "check" : Bool = PLC check AT %I2.4, 1 s
   "conv_broken" : Bool = PLC SIM_CV101 AT %M24.4, 1 s
   "conv_error" : Bool = PLC ALM_XA101_CV101 AT %M24.0, 1 s
   "CV-101" : Bool = PLC "CV-101" AT %Q4.0, 1 s
   "emergency" : Bool = PLC HMI_ES101 AT %M6.2, 1 s
   "FAN" : Bool = PLC "FN-101" AT %M11.3, 1 s
   "fan_broken" : Bool = PLC SIM_FN101 AT %M24.7, 1 s
   "fan_error" : Bool = PLC ALM_XA102_FN101 AT %M24.3, 1 s
   "HMI_FN101_Visible1" : Bool = PLC HMI_FN101_Visible1 AT %Q1.1, 1 s
   "HMI_FN101_Visible2" : Bool = PLC HMI_FN101_Visible2 AT %Q1.2, 1 s
   "HMI_Main" : Bool = PLC HMI_Main AT %M7.4, 1 s
   "HMI_PB_CV101" : Bool = PLC HMI_PB_CV101 AT %M8.2, 1 s
   "HMI_PB_FN101" : Bool = PLC HMI_PB_FN101 AT %M8.1, 1 s
   "HMI_PB_RB101" : Bool = PLC HMI_PB_RB101 AT %M7.7, 1 s
   "HMI_PB_RB102" : Bool = PLC HMI_PB_RB102 AT %M8.0, 1 s
   "HMI_PID" : Bool = PLC HMI_PID AT %M7.5, 1 s
   "HMI_RB102_Visible" : Bool = PLC HMI_RB102_Visible AT %Q1.4, 1 s
   "HMI_Status" : Bool = PLC HMI_Status AT %M7.6, 1 s
   "HMI_WP101_Visible" : Bool = PLC HMI_WP101_Visible AT %M7.0, 1 s
   "HMI_WP102_Visible" : Bool = PLC HMI_WP102_Visible AT %M7.1, 1 s
   "HMI_WP103_Visible" : Bool = PLC HMI_WP103_Visible AT %M7.2, 1 s
   "HMI_WP104_Visible" : Bool = PLC HMI_WP104_Visible AT %M7.3, 1 s
   "manip1_broken" : Bool = PLC SIM_RB101 AT %M24.5, 1 s
   "manip1_error" : Bool = PLC ALM_XA103_RB101 AT %M24.1, 1 s
   "manip2_broken" : Bool = PLC SIM_RB102 AT %M24.6, 1 s
   "manip2_error" : Bool = PLC ALM_XA104_RB102 AT %M24.2, 1 s
   "manu" : Bool = PLC HMI_PS104 AT %M6.4, 1 s
   "RB-101" : Bool = PLC "RB-101" AT %Q0.0, 1 s
   "RB-102" : Bool = PLC "RB-102" AT %Q0.2, 1 s
   "start" : Bool = PLC HMI_PS101 AT %M6.0, 1 s
   "stop" : Bool = PLC HMI_PS102 AT %M6.1, 1 s
   "ZS-101" : Bool = PLC "ZS-101" AT %I29.0, 1 s
   "ZS-102" : Bool = PLC "ZS-102" AT %I29.1, 1 s
   "ZS-103" : Bool = PLC "ZS-103" AT %I29.2, 1 s
   "ZS-104" : Bool = PLC "ZS-104" AT %I29.3, 1 s

discrete alarms
   8: 'Manipulator 2 is in tech-service.', class Warnings, trigger "Alarm_Collection" bit 7
   1: 'Something is wrong with the conveyor!!!', class Errors, trigger "Alarm_Collection" bit 0
   2: 'Conveyor is in tech-service.', class Warnings, trigger "Alarm_Collection" bit 1
   3: 'Something is wrong with the Manipulator 1!!!', class Errors, trigger "Alarm_Collection" bit 2
   4: 'Manipulator 1 is in tech-service.', class Warnings, trigger "Alarm_Collection" bit 3
   5: 'Something is wrong with the Fan!!!', class Errors, trigger "Alarm_Collection" bit 4
   6: 'Fan is in tech-service.', class Warnings, trigger "Alarm_Collection" bit 5
   7: 'Something is wrong with the Manipulator 2!!!', class Errors, trigger "Alarm_Collection" bit 6

text list "OFF_ON_LIST": 0 ''; 1 ''

screen "Error_Status" 800x420
   AlarmView "Alarm view_1" at 93,10 size 432x266
   Button "Button_17" at 578,66 size 140x17; TextOff 'ALM_XA101_ConveyorFault'
      on Press: function_b3f726e6("Alarm_Collection", 0); SetBit("conv_error")
   Button "Button_18" at 600,159 size 100x17; TextOff 'SIM_CV101_Broken'
      on Press: function_b3f726e6("Alarm_Collection", 1); SetBit("conv_broken")
   Button "Button_20" at 578,113 size 140x17; TextOff 'ALM_XA103_RB101Fault'
      on Press: function_b3f726e6("Alarm_Collection", 2); SetBit("manip1_error")
   Button "Button_22" at 600,206 size 100x17; TextOff 'SIM_RB101_Broken'
      on Press: function_b3f726e6("Alarm_Collection", 3); SetBit("manip1_broken")
   Button "Button_19" at 579,89 size 140x17; TextOff 'ALM_XA102_FanFault'
      on Press: function_b3f726e6("Alarm_Collection", 4); SetBit("fan_error")
   Button "Button_23" at 600,183 size 100x17; TextOff 'SIM_FN101_Broken'
      on Press: function_b3f726e6("Alarm_Collection", 5); SetBit("fan_broken")
   Button "Button_24" at 578,136 size 140x17; TextOff 'ALM_XA104_RB102Fault'
      on Press: function_b3f726e6("Alarm_Collection", 6); SetBit("manip2_error")
   Button "Button_25" at 600,229 size 100x17; TextOff 'SIM_RB102_Broken'
      on Press: function_b3f726e6("Alarm_Collection", 7); SetBit("manip2_broken")
   Button "Button_7" at 600,253 size 100x17; TextOff 'Repair all'
      on Press: function_a9b64e44("Alarm_Collection", 0); function_a9b64e44("Alarm_Collection", 1); function_a9b64e44("Alarm_Collection", 2); function_a9b64e44("Alarm_Collection", 3); function_a9b64e44("Alarm_Collection", 4); function_a9b64e44("Alarm_Collection", 5); function_a9b64e44("Alarm_Collection", 6); function_a9b64e44("Alarm_Collection", 7); ResetBit("conv_error"); ResetBit("conv_broken"); ResetBit("manip1_error"); ResetBit("manip1_broken"); ResetBit("fan_error"); ResetBit("fan_broken"); ResetBit("manip2_error"); ResetBit("manip2_broken")
   TextField "Text field_10" at 609,10 size 12x15; Text 'Text'
   Button "Button_1" at 541,10 size 217x17; TextOff 'ERROR STATUS'
      on Press: SetBit("HMI_Status")
      Appearance <- "HMI_Status"
   Button "Button_8" at 541,26 size 217x17; TextOff 'PID'
      on Press: ResetBit("HMI_Status"); ActivateScreen("PID", 0)
      Visibility <- "HMI_Status"
   Button "Button_9" at 541,43 size 217x17; TextOff 'CONTROL PANEL'
      on Press: ResetBit("HMI_Status"); ActivateScreen("Main Part", 0)
      Visibility <- "HMI_Status"

screen "Main Part" 800x420
   Circle "Circle_6" at 87,280 size 16x16
      Appearance <- "RB-101"
   IOField "I/O field_1" at 435,278 size 59x15; FormatPattern s99999
      ProcessValue <- "amount"
   Circle "Circle_7" at 425,83 size 16x16
      Appearance <- "RB-102"
   TextField "Text field_1" at 108,303 size 50x16; Text 'RB-101'
   TextField "Text field_2" at 230,275 size 49x16; Text 'FN-101'
   TextField "Text field_3" at 444,300 size 49x16; Text 'QI-101'
   TextField "Text field_4" at 442,64 size 50x16; Text 'RB-102'
   TextField "Text field_6" at 45,61 size 51x17; Text 'ZS-101'
   TextField "Text field_5" at 106,61 size 51x17; Text 'ZS-102'
   TextField "Text field_7" at 160,61 size 51x17; Text 'ZS-103'
   TextField "Text field_8" at 331,62 size 51x17; Text 'ZS-104'
   Button "Button_2" at 549,68 size 77x24; TextOff 'Start'; TextList "OFF_ON_LIST"
      on Press: SetBit("start"); ResetBit("stop")
      ProcessValue <- "start"
   Button "Button_6" at 549,103 size 77x24; TextOff 'STOP'
      on Press: SetBit("stop"); ResetBit("start")
      on Release: ResetBit("stop")
   GraphicView "Graphic view_2" at 152,280 size 20x18; Picture "Graphic_7"
      Visibility <- "manip1_broken"
   GraphicView "Graphic view_3" at 118,280 size 20x18; Picture "Graphic_8"
      Visibility <- "manip1_error"
   GraphicView "Graphic view_5" at 484,83 size 20x18; Picture "Graphic_7"
      Appearance <- "manip2_broken"
   GraphicView "Graphic view_7" at 454,82 size 20x18; Picture "Graphic_8"
      Appearance <- "manip2_error"
   Circle "Circle_16" at 59,83 size 11x11
      Appearance <- "ZS-101"
   Circle "Circle_18" at 120,82 size 11x11
      Appearance <- "ZS-102"
   Circle "Circle_20" at 306,190 size 16x16
      Appearance <- "CV-101"
   GraphicView "Graphic view_1" at 336,190 size 20x18; Picture "Graphic_8"
      Appearance <- "conv_error"
   GraphicView "Graphic view_8" at 365,190 size 20x18; Picture "Graphic_7"
      Appearance <- "conv_broken"
   TextField "Text field_11" at 329,212 size 50x16; Text 'CV-101'
   Circle "Circle_8" at 184,82 size 11x11
      Appearance <- "ZS-103"
   Circle "Circle_9" at 347,81 size 11x11
      Appearance <- "ZS-104"
   Rectangle "Rectangle_15" at 444,128 size 31x55
      Visibility <- "HMI_RB102_Visible"
   Rectangle "Rectangle_18" at 451,184 size 20x42
      Visibility <- "HMI_RB102_Visible"
   Rectangle "Rectangle_19" at 448,226 size 26x9
      Visibility <- "HMI_RB102_Visible"
   Group "Group" at 52,118 size 44x38
   Circle "Circle_11" at 211,254 size 16x16
      Appearance <- "FAN"
   GraphicView "Graphic view_4" at 266,253 size 20x18; Picture "Graphic_7"
      Appearance <- "fan_broken"
   GraphicView "Graphic view_6" at 239,253 size 20x18; Picture "Graphic_8"
      Appearance <- "fan_error"
   Circle "Circle_13" at 696,211 size 35x35
      Appearance <- "emergency"
   Button "Button_12" at 551,216 size 77x24; TextOff 'Emergency'
      on Press: SetBit("emergency"); ResetBit("start"); ResetBit("auto"); ResetBit("manu")
      on Release: ResetBit("emergency")
   Button "Button_1" at 548,171 size 77x24; TextOff 'Auto Mode'
      on Press: SetBit("auto"); ResetBit("manu")
   Button "Button_13" at 549,138 size 77x24; TextOff 'Manu Mode'
      on Press: SetBit("manu"); ResetBit("auto")
   Button "Button_14" at 668,68 size 77x24; TextOff 'PB_RB101'
      on Press: SetBit("HMI_PB_RB101")
      on Release: ResetBit("HMI_PB_RB101")
   Button "Button_3" at 668,135 size 77x24; TextOff 'PB_RB102'
      on Press: SetBit("HMI_PB_RB102")
      on Release: ResetBit("HMI_PB_RB102")
   Button "Button_4" at 668,101 size 77x24; TextOff 'PB_FN101'
      on Press: SetBit("HMI_PB_FN101")
      on Release: ResetBit("HMI_PB_FN101")
   Button "Button_5" at 668,167 size 77x24; TextOff 'PB_CV101'
      on Press: SetBit("HMI_PB_CV101")
      on Release: ResetBit("HMI_PB_CV101")
   GraphicView "Graphic view_15" at 118,280 size 20x18; Picture "Graphic_10"
      Visibility <- "manip1_error"
   GraphicView "Graphic view_16" at 152,280 size 20x18; Picture "Graphic_9"
      Visibility <- "manip1_broken"
   GraphicView "Graphic view_17" at 239,253 size 20x18; Picture "Graphic_10"
      Visibility <- "fan_error"
   GraphicView "Graphic view_18" at 266,253 size 20x18; Picture "Graphic_9"
      Visibility <- "fan_broken"
   GraphicView "Graphic view_19" at 365,190 size 20x18; Picture "Graphic_9"
      Visibility <- "conv_broken"
   GraphicView "Graphic view_20" at 336,190 size 20x18; Picture "Graphic_10"
      Visibility <- "conv_error"
   GraphicView "Graphic view_21" at 454,82 size 20x18; Picture "Graphic_10"
      Visibility <- "manip2_error"
   GraphicView "Graphic view_22" at 484,83 size 20x18; Picture "Graphic_9"
      Visibility <- "manip2_broken"
   TextField "Text field_10" at 609,10 size 12x15; Text 'Text'
   Button "Button_7" at 541,10 size 217x17; TextOff 'CONTROL PANEL'
      on Press: SetBit("HMI_Main")
      Appearance <- "HMI_Main"
   Button "Button_8" at 541,26 size 217x17; TextOff 'PID'
      on Press: ResetBit("HMI_Main"); ActivateScreen("PID", 0)
      Visibility <- "HMI_Main"
   Button "Button_9" at 541,43 size 217x17; TextOff 'ERROR STATUS'
      on Press: ResetBit("HMI_Main"); ActivateScreen("Error_Status", 0)
      Visibility <- "HMI_Main"
   Group "Group_1" at 109,118 size 44x38
   Group "Group_2" at 191,118 size 44x38
   Group "Group_3" at 341,119 size 44x38
   Rectangle "Rectangle_22" at 417,128 size 59x28
      Visibility <- "HMI_RB102_Visible"
   Rectangle "Rectangle_23" at 371,132 size 46x18
      Visibility <- "HMI_RB102_Visible"
   Rectangle "Rectangle_24" at 361,130 size 10x24
      Visibility <- "HMI_RB102_Visible"
   GraphicView "Graphic view_9" at 223,77 size 52x49; Picture "Graphic_14"
      Visibility <- "FAN"
   GraphicView "Graphic view_10" at 223,77 size 52x49; Picture "Graphic_15"
      Visibility <- "HMI_FN101_Visible1"
   GraphicView "Graphic view_11" at 223,137 size 52x49; Picture "Graphic_14"
   GraphicView "Graphic view_12" at 223,137 size 52x49; Picture "Graphic_15"
      Visibility <- "HMI_FN101_Visible1"
   GraphicView "Graphic view_13" at 223,77 size 52x49; Picture "Graphic_16"
      Visibility <- "HMI_FN101_Visible2"
   GraphicView "Graphic view_14" at 223,137 size 52x49; Picture "Graphic_16"
      Visibility <- "HMI_FN101_Visible2"
   TextField "Text field_12" at 694,247 size 48x16; Text 'ES-101'
   Rectangle "Rectangle_44" at 52,118 size 44x29
      Appearance <- "block_color"
      Visibility <- "HMI_WP101_Visible"
   Rectangle "Rectangle_45" at 52,147 size 44x10
      Appearance <- "block_color"
      Visibility <- "HMI_WP101_Visible"
   Rectangle "Rectangle_31" at 109,118 size 44x29
      Appearance <- "block_color"
      Visibility <- "HMI_WP102_Visible"
   Rectangle "Rectangle_32" at 109,147 size 44x10
      Appearance <- "block_color"
      Visibility <- "HMI_WP102_Visible"
   Rectangle "Rectangle_33" at 191,118 size 44x29
      Appearance <- "block_color"
      Visibility <- "HMI_WP103_Visible"
   Rectangle "Rectangle_34" at 191,147 size 44x10
      Appearance <- "block_color"
      Visibility <- "HMI_WP103_Visible"
   Rectangle "Rectangle_35" at 341,119 size 44x29
      Appearance <- "block_color"
      Visibility <- "HMI_WP104_Visible"
   Rectangle "Rectangle_46" at 341,147 size 44x10
      Appearance <- "block_color"
      Visibility <- "HMI_WP104_Visible"

screen "PID" 800x420
   TextField "Text field_10" at 609,10 size 12x15; Text 'Text'
   Button "Button_1" at 541,10 size 217x17; TextOff 'PID'
      on Press: SetBit("HMI_PID")
      Appearance <- "HMI_PID"
   Button "Button_8" at 541,26 size 217x17; TextOff 'ERROR STATUS'
      on Press: ResetBit("HMI_PID"); ActivateScreen("Error_Status", 0)
      Visibility <- "HMI_PID"
   Button "Button_9" at 541,43 size 217x17; TextOff 'CONTROL PANEL'
      on Press: ResetBit("HMI_PID"); ActivateScreen("Main Part", 0)
      Visibility <- "HMI_PID"
   TrendView "Trend view_1" at 93,10 size 432x266
   IOField "I/O field_1" at 688,75 size 59x15; FormatPattern s99999
      ProcessValue <- "amount"
   IOField "I/O field_2" at 688,102 size 59x15; FormatPattern s99999
      ProcessValue <- "amount"
   IOField "I/O field_3" at 688,128 size 59x15; FormatPattern s99999
      ProcessValue <- "amount"
   IOField "I/O field_4" at 688,155 size 59x15; FormatPattern s99999
      ProcessValue <- "amount"
   TextField "Text field_4" at 634,75 size 54x16; Text 'Setpoint'
   TextField "Text field_1" at 658,102 size 27x16; Text 'K_p'
   TextField "Text field_2" at 658,128 size 24x16; Text 'K_i'
   TextField "Text field_3" at 658,155 size 27x16; Text 'K_d'
   Rectangle "Rectangle_22" at 551,80 size 70x85
      Visibility <- "HMI_RB102_Visible"
   Circle "Circle_13" at 590,88 size 24x24
      Appearance <- "emergency"
   Circle "Circle_1" at 590,131 size 24x24
      Appearance <- "emergency"
   TextField "Text field_5" at 555,92 size 35x16; Text 'Start'
   TextField "Text field_6" at 556,135 size 31x16; Text 'Stop'
*)